// TIA Portal V20 export
DATA_BLOCK "GLOBAL_PROCESS_STOP_HMI_IF_DB"   // DB213
{ S7_Optimized_Access := 'TRUE' }
// stored: AutoNumber false, MemoryReserve 100
   VAR
      PROCESS_STOP { S7_SetPoint := 'True'} : Array[0..5] of "MISC_PROCESS_STOP_HMI_UDT";
   END_VAR
BEGIN
   // PROCESS_STOP[1] : +ST020-TL01
   // PROCESS_STOP[2] : +ST025-TL01
   // PROCESS_STOP[3] : +ST025-TL02
   // PROCESS_STOP[4] : +ST030-TL01
END_DATA_BLOCK
